ABB RobotStudio station: ⁭ifmm_solution.rspag

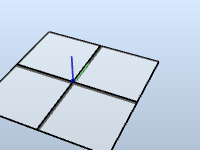
Station Solution2 (saved by RobotStudio 6.4.7120.133)
Layout (positions relative to the parent item):
